{attribute 'qualified_only'}
{attribute 'strict'}
{attribute 'to_string'}
TYPE eRobPosType :
(
	Absolut := 0,			// Absolute Bewegung bezogen auf Basis-Koordinatensystem
	Relativ := 1			// Relative Bewegung bezogen auf aktuelle Position
);
END_TYPE

(* stored: Version 1.1.0.1
   DUT eRobPosType: Id {e7690974-672a-40ec-a33a-3474c076613c} *)
